// TIA Portal V19 export
VAR_GLOBAL   // PLC tag table "SlurryIOs"
END_VAR
